FUNCTION_BLOCK FB_Enabled IMPLEMENTS I_State
VAR_INPUT
END_VAR
VAR_OUTPUT
END_VAR
VAR
	pAxis : POINTER TO FB_Axis;
END_VAR

{warning 'add method implementation '}
METHOD Disable : BOOL

VAR
END_VAR
ADSLOGSTR(ADSLOG_MSGTYPE_HINT, 'user has disabled.', '');
pAxis^.SetState(pAxis^.IdleState);
END_METHOD

{warning 'add method implementation '}
METHOD Enable : BOOL
END_METHOD

METHOD FB_init : BOOL
VAR_INPUT
	bInitRetains : BOOL; // if TRUE, the retain variables are initialized (warm start / cold start)
	bInCopyCode : BOOL;  // if TRUE, the instance afterwards gets moved into the copy code (online change)
	pAxis : POINTER TO FB_Axis;
END_VAR
THIS^.pAxis := pAxis;
END_METHOD

{warning 'add method implementation '}
METHOD Reset : BOOL
END_METHOD

{warning 'add property implementation'}
PROPERTY State : STRING
GET
State := 'Enabled';
END_GET
END_PROPERTY

END_FUNCTION_BLOCK

(* stored: Version 1.1.0.1, ProductVersion 3.1.4024.3
   POU FB_Enabled: Id {175046d5-4c37-4314-a67d-9b219422be85}, SpecialFunc None
   Method Disable: Id {44772350-f6a9-4090-868b-7247c661a587}
   Method Enable: Id {cf1e48b2-d807-4f0a-9199-df346117d3f4}
   Method FB_init: Id {f8a6feec-166a-4acb-b8dc-94f59db25dcd}
   Method Reset: Id {d8f93f58-4cbc-4d04-b4d0-b4f84387d0e2}
   Property State: Id {0750bc65-a466-4335-adf8-2efeceefab1e}
   Get Get: Id {f9cd22f6-1fa0-4012-bf0a-f8c2035c7e79} *)
